TYPE ST_CardState_HWI :
STRUCT
  uiDataState   : UINT;
  bWcState      : BOOL := FALSE;
END_STRUCT
END_TYPE

(* stored: Version 1.1.0.1, ProductVersion 3.1.4024.12
   DUT ST_CardState_HWI: Id {a1b089d7-5221-402c-872a-306d83b3a3d0} *)
